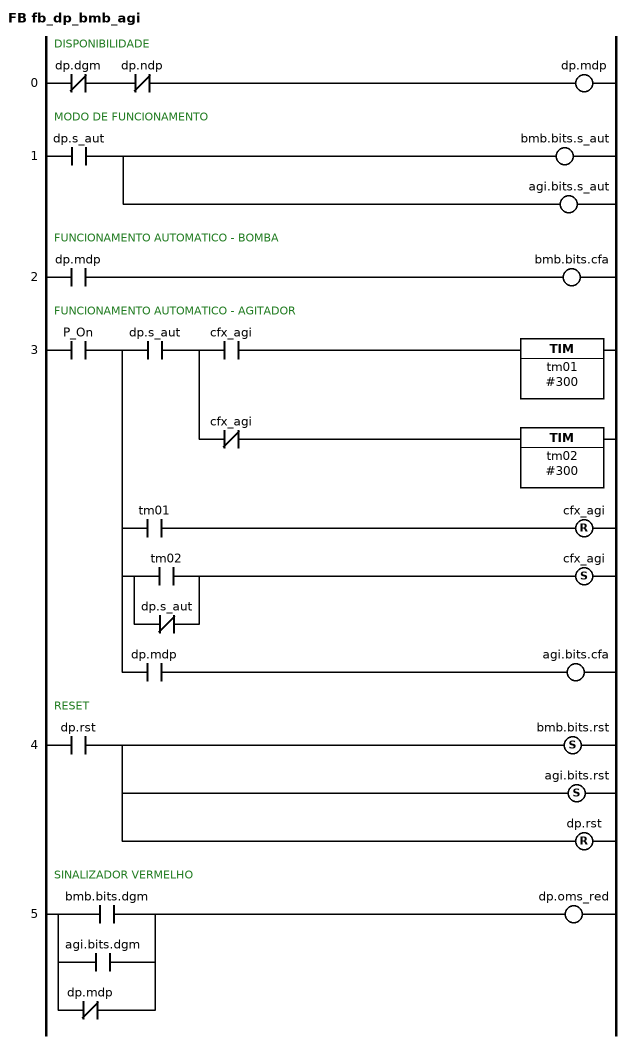
; [picture p24: FB fb_dp_bmb_agi, rungs 0-5]
; rung 0: DISPONIBILIDADE
LDNOT dp.dgm
ANDNOT dp.ndp
OUT dp.mdp
; rung 1: MODO DE FUNCIONAMENTO
LD dp.s_aut
OUT bmb.bits.s_aut
OUT agi.bits.s_aut
; rung 2: FUNCIONAMENTO AUTOMATICO - BOMBA
LD dp.mdp
OUT bmb.bits.cfa
; rung 3: FUNCIONAMENTO AUTOMATICO - AGITADOR
LD P_On
OUT TR0
AND dp.s_aut
OUT TR1
AND cfx_agi
TIM tm01 #300
LD TR1
ANDNOT cfx_agi
TIM tm02 #300
LD TR0
AND tm01
RSET cfx_agi
LD TR0
LD tm02
ORNOT dp.s_aut
ANDLD
SET cfx_agi
LD TR0
AND dp.mdp
OUT agi.bits.cfa
; rung 4: RESET
LD dp.rst
SET bmb.bits.rst
SET agi.bits.rst
RSET dp.rst
; rung 5: SINALIZADOR VERMELHO
LD bmb.bits.dgm
OR agi.bits.dgm
ORNOT dp.mdp
OUT dp.oms_red

## Function block fb_dp_pss_agi_vlv
; FUNÇÃO DEPOSITO DE PRODUTO COM PRESSORIZAÇÃO/AGITADOR/VALVULA - Executa o funcionamento de um deposito de produto constituido por pressorização, um agitador e uma valvula.
VAR_IN_OUT
  dp : s_deposito_p;  (* Dados do deposito *)
  pss : s_equip;  (* Dados da pressorização *)
  agi : s_equip;  (* Dados do agitador *)
  vlv : s_equip;  (* Dados da válvula *)
END_VAR
VAR
  tm01 : TIMER;
  tm02 : TIMER;
  cfx_agi : BOOL;
END_VAR

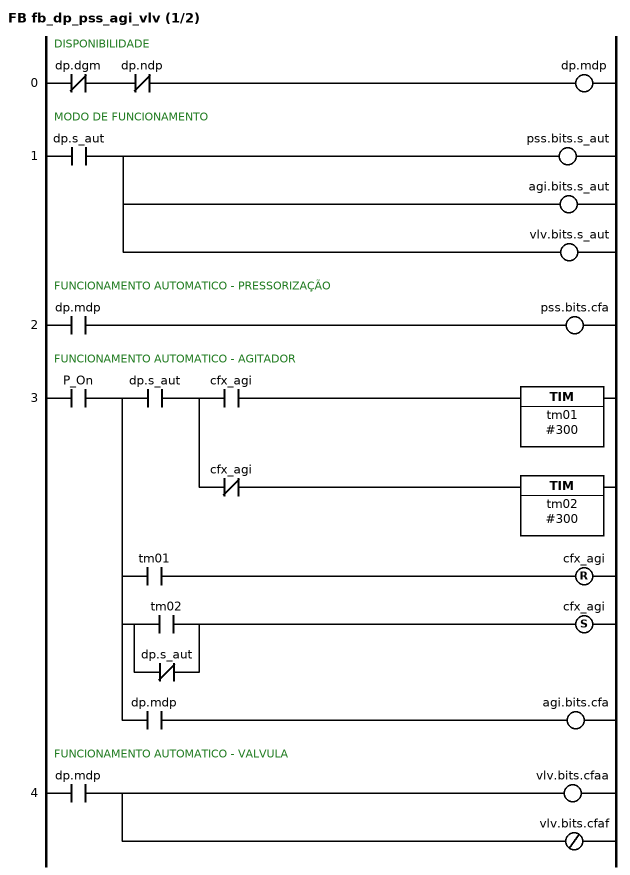
; rung 0: DISPONIBILIDADE
LDNOT dp.dgm
ANDNOT dp.ndp
OUT dp.mdp
; rung 1: MODO DE FUNCIONAMENTO
LD dp.s_aut
OUT pss.bits.s_aut
OUT agi.bits.s_aut
OUT vlv.bits.s_aut
; rung 2: FUNCIONAMENTO AUTOMATICO - PRESSORIZAÇÃO
LD dp.mdp
OUT pss.bits.cfa
; rung 3: FUNCIONAMENTO AUTOMATICO - AGITADOR
LD P_On
OUT TR0
AND dp.s_aut
OUT TR1
AND cfx_agi
TIM tm01 #300
LD TR1
ANDNOT cfx_agi
TIM tm02 #300
LD TR0
AND tm01
RSET cfx_agi
LD TR0
LD tm02
ORNOT dp.s_aut
ANDLD
SET cfx_agi
LD TR0
AND dp.mdp
OUT agi.bits.cfa
; rung 4: FUNCIONAMENTO AUTOMATICO - VALVULA
LD dp.mdp
OUT vlv.bits.cfaa
OUTNOT vlv.bits.cfaf

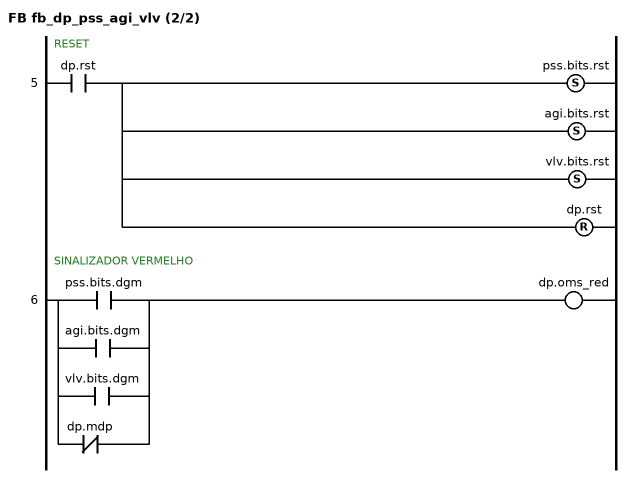
; rung 5: RESET
LD dp.rst
SET pss.bits.rst
SET agi.bits.rst
SET vlv.bits.rst
RSET dp.rst
; rung 6: SINALIZADOR VERMELHO
LD pss.bits.dgm
OR agi.bits.dgm
OR vlv.bits.dgm
ORNOT dp.mdp
OUT dp.oms_red

## Function block fb_eq_bomba
; FUNÇÃO BOMBA - Controlo de uma maquina tipo bomba.
VAR_IN_OUT
  bmb : s_equip;  (* Dados do motor *)
END_VAR
VAR
  tm01 : TIMER;
  tm02 : TIMER;
  ct01 : COUNTER;
  tm_b_x : DINT;
END_VAR

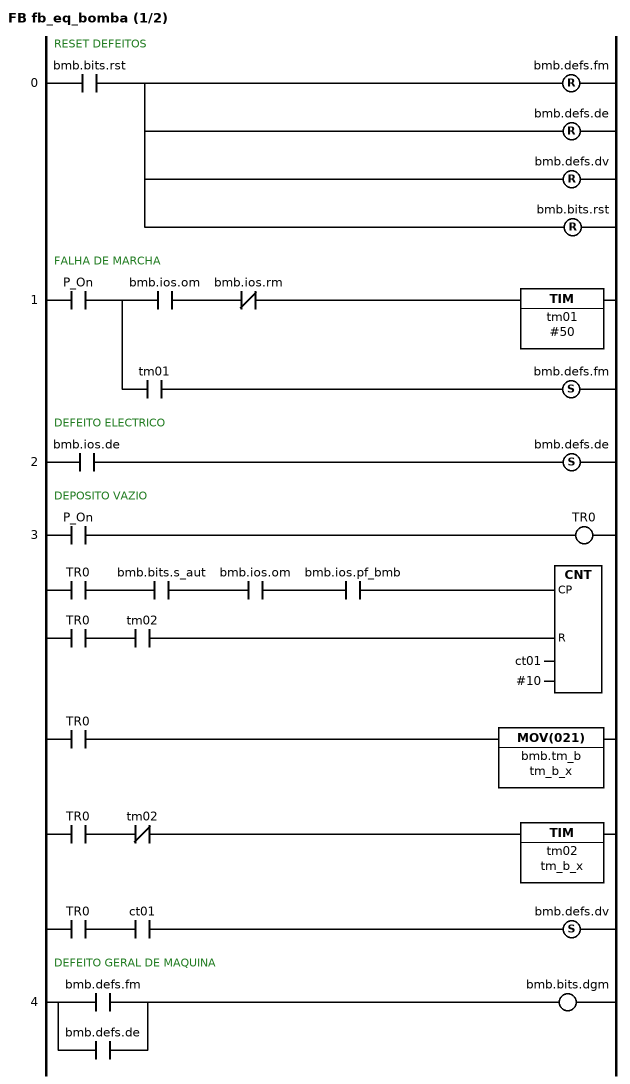
; rung 0: RESET DEFEITOS
LD bmb.bits.rst
RSET bmb.defs.fm
RSET bmb.defs.de
RSET bmb.defs.dv
RSET bmb.bits.rst
; rung 1: FALHA DE MARCHA
LD P_On
OUT TR0
AND bmb.ios.om
ANDNOT bmb.ios.rm
TIM tm01 #50
LD TR0
AND tm01
SET bmb.defs.fm
; rung 2: DEFEITO ELECTRICO
LD bmb.ios.de
SET bmb.defs.de
; rung 3: DEPOSITO VAZIO
LD P_On
OUT TR0
LD TR0
AND bmb.bits.s_aut
AND bmb.ios.om
AND bmb.ios.pf_bmb
LD TR0
AND tm02
CNT ct01 #10
LD TR0
MOV(021) bmb.tm_b tm_b_x
LD TR0
ANDNOT tm02
TIM tm02 tm_b_x
LD TR0
AND ct01
SET bmb.defs.dv
; rung 4: DEFEITO GERAL DE MAQUINA
LD bmb.defs.fm
OR bmb.defs.de
OUT bmb.bits.dgm

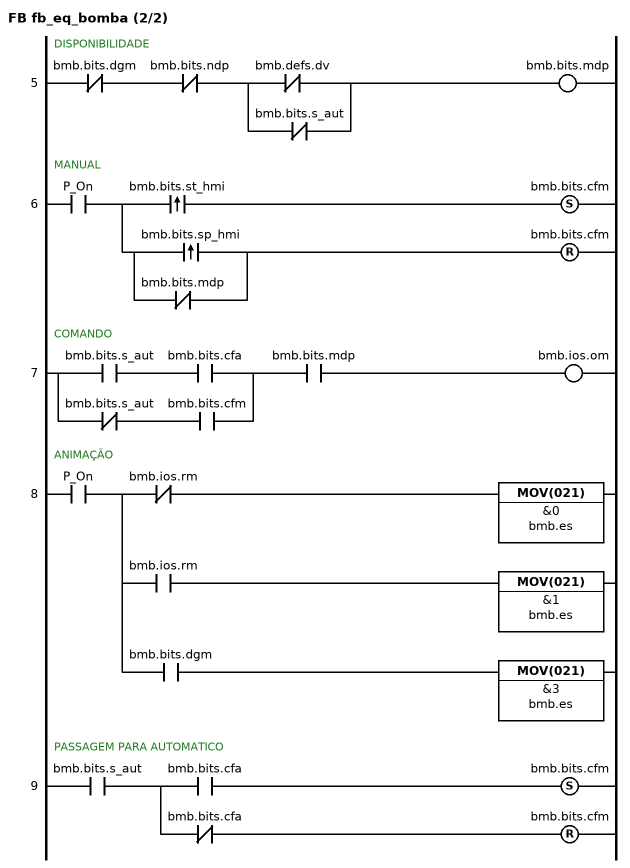
; rung 5: DISPONIBILIDADE
LDNOT bmb.bits.dgm
ANDNOT bmb.bits.ndp
LDNOT bmb.defs.dv
ORNOT bmb.bits.s_aut
ANDLD
OUT bmb.bits.mdp
; rung 6: MANUAL
LD P_On
OUT TR0
@AND bmb.bits.st_hmi
SET bmb.bits.cfm
LD TR0
@LD bmb.bits.sp_hmi
ORNOT bmb.bits.mdp
ANDLD
RSET bmb.bits.cfm
; rung 7: COMANDO
LD bmb.bits.s_aut
AND bmb.bits.cfa
LDNOT bmb.bits.s_aut
AND bmb.bits.cfm
ORLD
AND bmb.bits.mdp
OUT bmb.ios.om
; rung 8: ANIMAÇÃO
LD P_On
OUT TR0
ANDNOT bmb.ios.rm
MOV(021) &0 bmb.es
LD TR0
AND bmb.ios.rm
MOV(021) &1 bmb.es
LD TR0
AND bmb.bits.dgm
MOV(021) &3 bmb.es
; rung 9: PASSAGEM PARA AUTOMATICO
LD bmb.bits.s_aut
OUT TR0
AND bmb.bits.cfa
SET bmb.bits.cfm
LD TR0
ANDNOT bmb.bits.cfa
RSET bmb.bits.cfm

## Function block fb_eq_motor
; FUNÇÃO MOTOR - Controlo de uma maquina tipo motor.
VAR_IN_OUT
  mot : s_equip;  (* Dados do motor *)
END_VAR
VAR
  tm01 : TIMER;
END_VAR

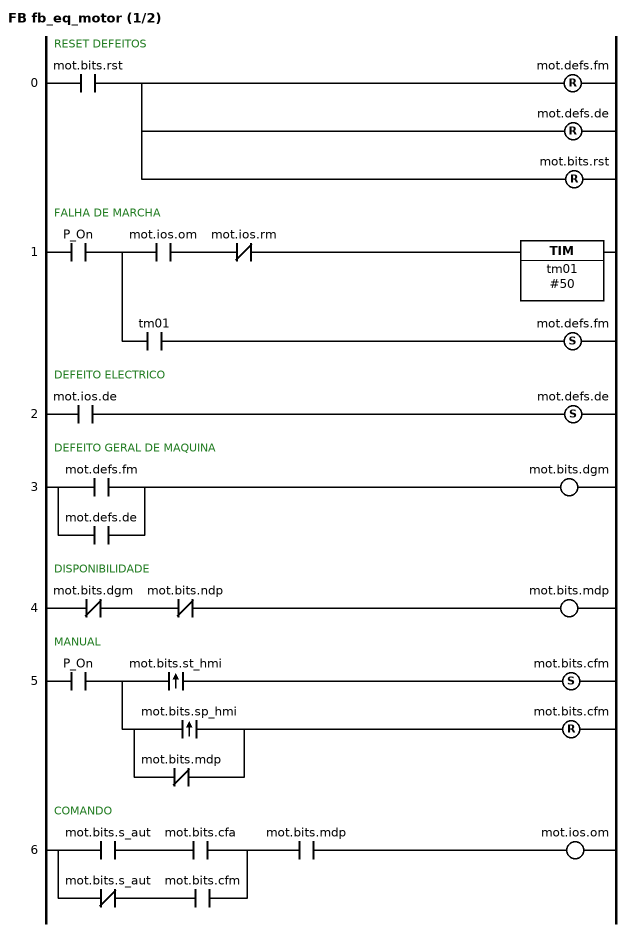
; rung 0: RESET DEFEITOS
LD mot.bits.rst
RSET mot.defs.fm
RSET mot.defs.de
RSET mot.bits.rst
; rung 1: FALHA DE MARCHA
LD P_On
OUT TR0
AND mot.ios.om
ANDNOT mot.ios.rm
TIM tm01 #50
LD TR0
AND tm01
SET mot.defs.fm
; rung 2: DEFEITO ELECTRICO
LD mot.ios.de
SET mot.defs.de
; rung 3: DEFEITO GERAL DE MAQUINA
LD mot.defs.fm
OR mot.defs.de
OUT mot.bits.dgm
; rung 4: DISPONIBILIDADE
LDNOT mot.bits.dgm
ANDNOT mot.bits.ndp
OUT mot.bits.mdp
; rung 5: MANUAL
LD P_On
OUT TR0
@AND mot.bits.st_hmi
SET mot.bits.cfm
LD TR0
@LD mot.bits.sp_hmi
ORNOT mot.bits.mdp
ANDLD
RSET mot.bits.cfm
; rung 6: COMANDO
LD mot.bits.s_aut
AND mot.bits.cfa
LDNOT mot.bits.s_aut
AND mot.bits.cfm
ORLD
AND mot.bits.mdp
OUT mot.ios.om

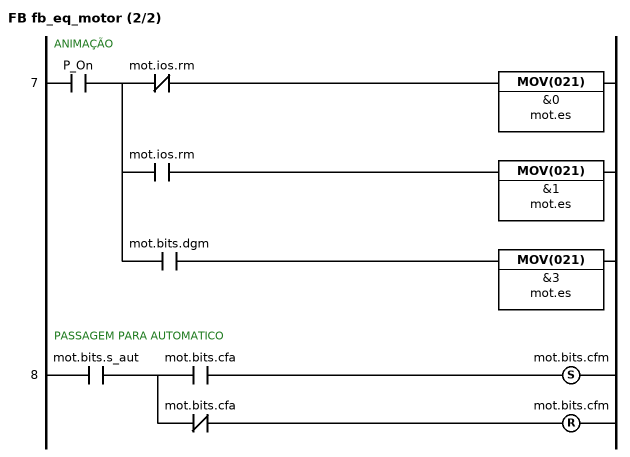
; rung 7: ANIMAÇÃO
LD P_On
OUT TR0
ANDNOT mot.ios.rm
MOV(021) &0 mot.es
LD TR0
AND mot.ios.rm
MOV(021) &1 mot.es
LD TR0
AND mot.bits.dgm
MOV(021) &3 mot.es
; rung 8: PASSAGEM PARA AUTOMATICO
LD mot.bits.s_aut
OUT TR0
AND mot.bits.cfa
SET mot.bits.cfm
LD TR0
ANDNOT mot.bits.cfa
RSET mot.bits.cfm

## Function block fb_eq_press
; FUNÇÃO PRESSORIZAR - Controlo de uma maquina tipo motor.
VAR_IN_OUT
  press : s_equip;  (* Dados da presseorização *)
END_VAR
VAR
  tm01 : TIMER;
END_VAR

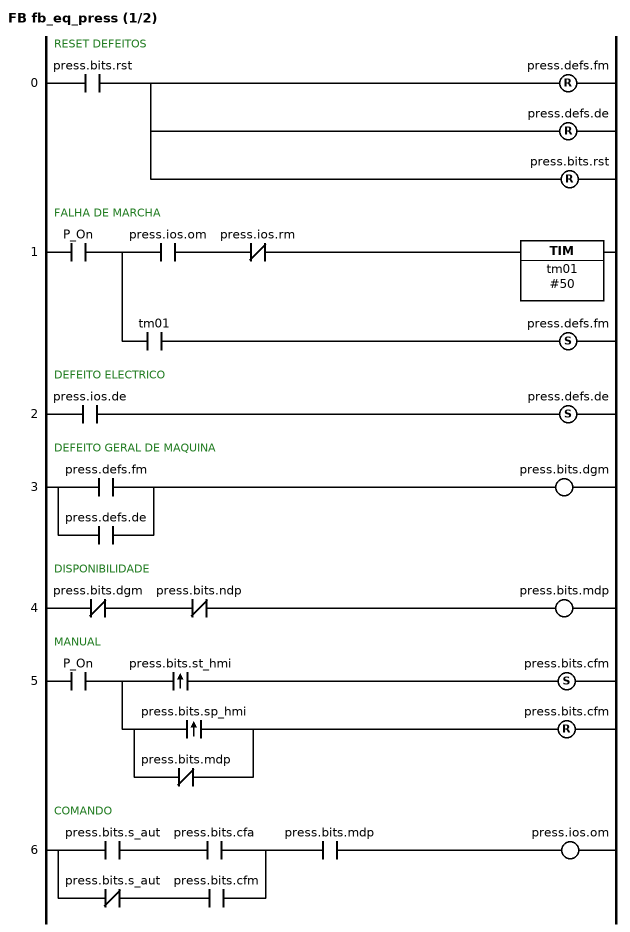
; rung 0: RESET DEFEITOS
LD press.bits.rst
RSET press.defs.fm
RSET press.defs.de
RSET press.bits.rst
; rung 1: FALHA DE MARCHA
LD P_On
OUT TR0
AND press.ios.om
ANDNOT press.ios.rm
TIM tm01 #50
LD TR0
AND tm01
SET press.defs.fm
; rung 2: DEFEITO ELECTRICO
LD press.ios.de
SET press.defs.de
; rung 3: DEFEITO GERAL DE MAQUINA
LD press.defs.fm
OR press.defs.de
OUT press.bits.dgm
; rung 4: DISPONIBILIDADE
LDNOT press.bits.dgm
ANDNOT press.bits.ndp
OUT press.bits.mdp
; rung 5: MANUAL
LD P_On
OUT TR0
@AND press.bits.st_hmi
SET press.bits.cfm
LD TR0
@LD press.bits.sp_hmi
ORNOT press.bits.mdp
ANDLD
RSET press.bits.cfm
; rung 6: COMANDO
LD press.bits.s_aut
AND press.bits.cfa
LDNOT press.bits.s_aut
AND press.bits.cfm
ORLD
AND press.bits.mdp
OUT press.ios.om

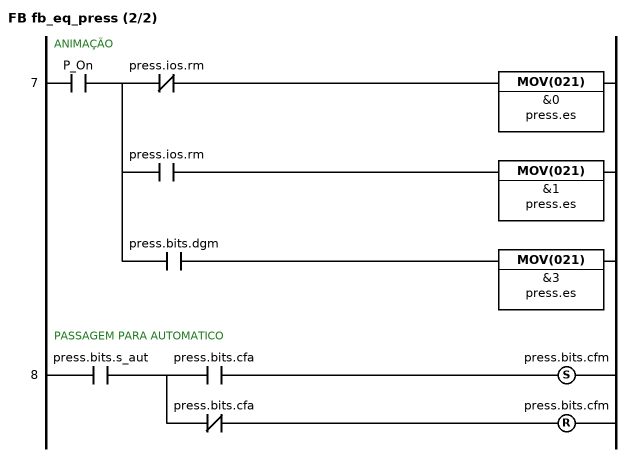
; rung 7: ANIMAÇÃO
LD P_On
OUT TR0
ANDNOT press.ios.rm
MOV(021) &0 press.es
LD TR0
AND press.ios.rm
MOV(021) &1 press.es
LD TR0
AND press.bits.dgm
MOV(021) &3 press.es
; rung 8: PASSAGEM PARA AUTOMATICO
LD press.bits.s_aut
OUT TR0
AND press.bits.cfa
SET press.bits.cfm
LD TR0
ANDNOT press.bits.cfa
RSET press.bits.cfm

## Function block fb_eq_valvula
; FUNÇÃO VALVULA - Controlo de uma maquina tipo valvula.
VAR_IN_OUT
  valv : s_equip;  (* Dados da valvula *)
END_VAR
VAR
  tm01 : TIMER;
  tm02 : TIMER;
END_VAR

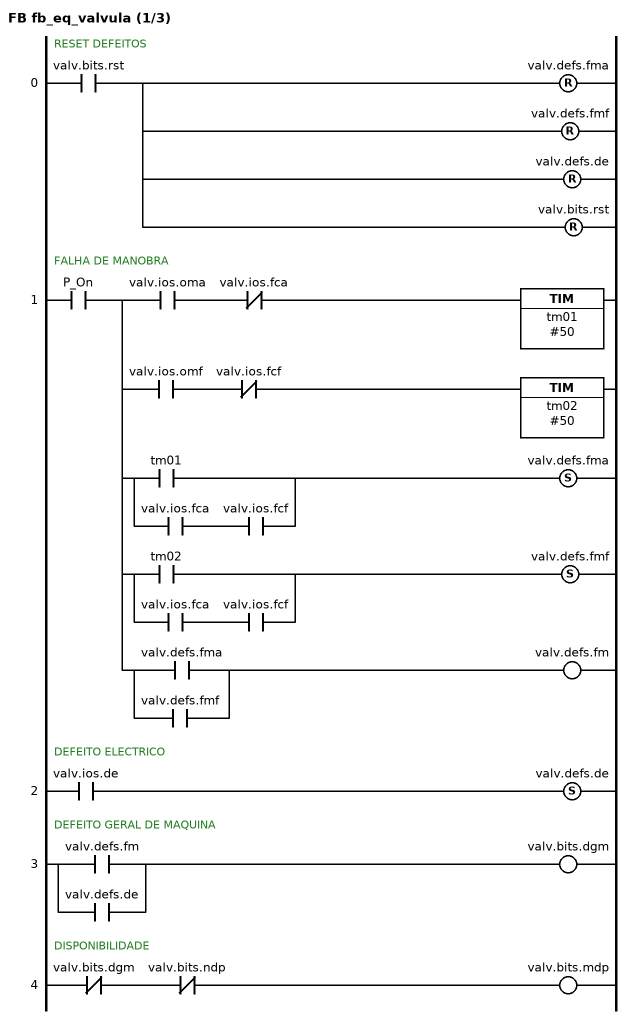
; rung 0: RESET DEFEITOS
LD valv.bits.rst
RSET valv.defs.fma
RSET valv.defs.fmf
RSET valv.defs.de
RSET valv.bits.rst
; rung 1: FALHA DE MANOBRA
LD P_On
OUT TR0
AND valv.ios.oma
ANDNOT valv.ios.fca
TIM tm01 #50
LD TR0
AND valv.ios.omf
ANDNOT valv.ios.fcf
TIM tm02 #50
LD TR0
LD tm01
LD valv.ios.fca
AND valv.ios.fcf
ORLD
ANDLD
SET valv.defs.fma
LD TR0
LD tm02
LD valv.ios.fca
AND valv.ios.fcf
ORLD
ANDLD
SET valv.defs.fmf
LD TR0
LD valv.defs.fma
OR valv.defs.fmf
ANDLD
OUT valv.defs.fm
; rung 2: DEFEITO ELECTRICO
LD valv.ios.de
SET valv.defs.de
; rung 3: DEFEITO GERAL DE MAQUINA
LD valv.defs.fm
OR valv.defs.de
OUT valv.bits.dgm
; rung 4: DISPONIBILIDADE
LDNOT valv.bits.dgm
ANDNOT valv.bits.ndp
OUT valv.bits.mdp

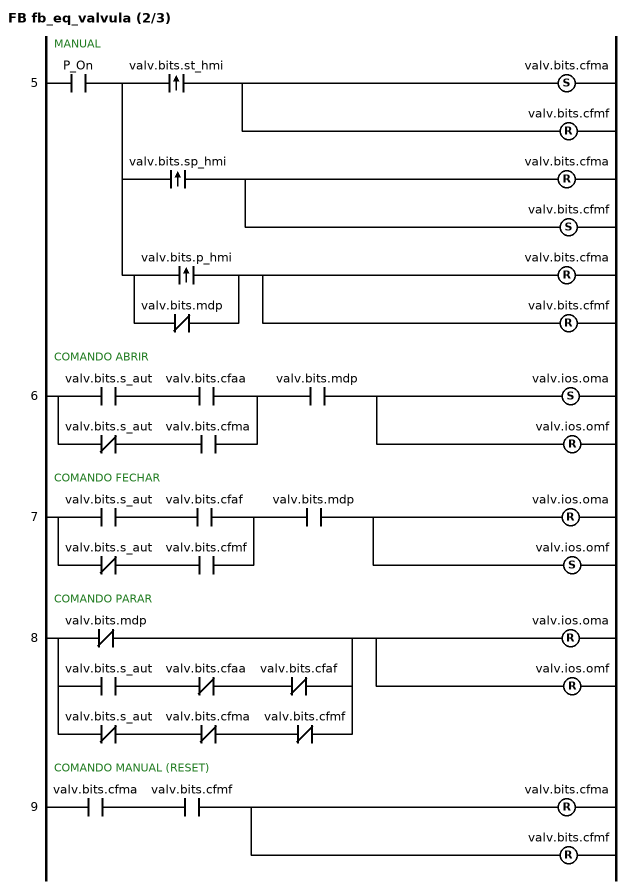
; rung 5: MANUAL
LD P_On
OUT TR0
@AND valv.bits.st_hmi
SET valv.bits.cfma
RSET valv.bits.cfmf
LD TR0
@AND valv.bits.sp_hmi
RSET valv.bits.cfma
SET valv.bits.cfmf
LD TR0
@LD valv.bits.p_hmi
ORNOT valv.bits.mdp
ANDLD
RSET valv.bits.cfma
RSET valv.bits.cfmf
; rung 6: COMANDO ABRIR
LD valv.bits.s_aut
AND valv.bits.cfaa
LDNOT valv.bits.s_aut
AND valv.bits.cfma
ORLD
AND valv.bits.mdp
SET valv.ios.oma
RSET valv.ios.omf
; rung 7: COMANDO FECHAR
LD valv.bits.s_aut
AND valv.bits.cfaf
LDNOT valv.bits.s_aut
AND valv.bits.cfmf
ORLD
AND valv.bits.mdp
RSET valv.ios.oma
SET valv.ios.omf
; rung 8: COMANDO PARAR
LDNOT valv.bits.mdp
LD valv.bits.s_aut
ANDNOT valv.bits.cfaa
ANDNOT valv.bits.cfaf
ORLD
LDNOT valv.bits.s_aut
ANDNOT valv.bits.cfma
ANDNOT valv.bits.cfmf
ORLD
RSET valv.ios.oma
RSET valv.ios.omf
; rung 9: COMANDO MANUAL (RESET)
LD valv.bits.cfma
AND valv.bits.cfmf
RSET valv.bits.cfma
RSET valv.bits.cfmf

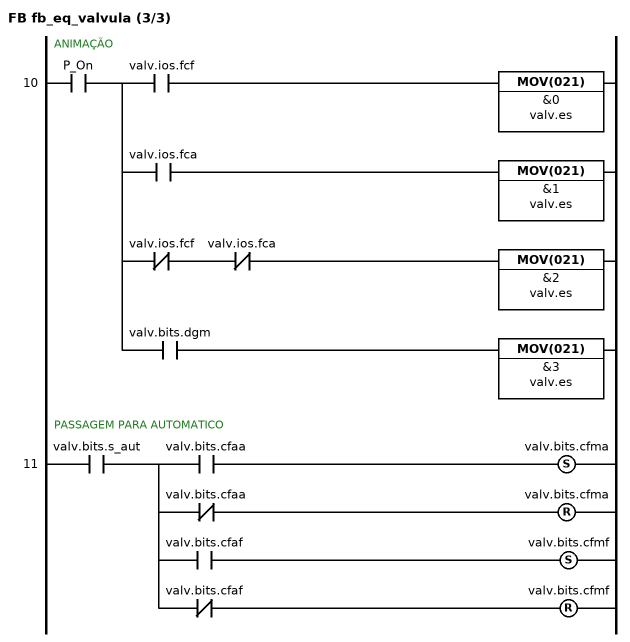
; rung 10: ANIMAÇÃO
LD P_On
OUT TR0
AND valv.ios.fcf
MOV(021) &0 valv.es
LD TR0
AND valv.ios.fca
MOV(021) &1 valv.es
LD TR0
ANDNOT valv.ios.fcf
ANDNOT valv.ios.fca
MOV(021) &2 valv.es
LD TR0
AND valv.bits.dgm
MOV(021) &3 valv.es
; rung 11: PASSAGEM PARA AUTOMATICO
LD valv.bits.s_aut
OUT TR0
AND valv.bits.cfaa
SET valv.bits.cfma
LD TR0
ANDNOT valv.bits.cfaa
RSET valv.bits.cfma
LD TR0
AND valv.bits.cfaf
SET valv.bits.cfmf
LD TR0
ANDNOT valv.bits.cfaf
RSET valv.bits.cfmf

## Function block fb_inj_caudal
; FUNÇÃO CAUDALIMETRO - Caudalimetro local/remoto
VAR_IN_OUT
  tt : s_caudal;  (* Dados do caudalímetro *)
END_VAR
VAR
  tt_rem_d : REAL;  (* Diferença de totalização *)
  tm01 : TIMER;
  tm02 : TIMER;
  ct01 : COUNTER;
END_VAR

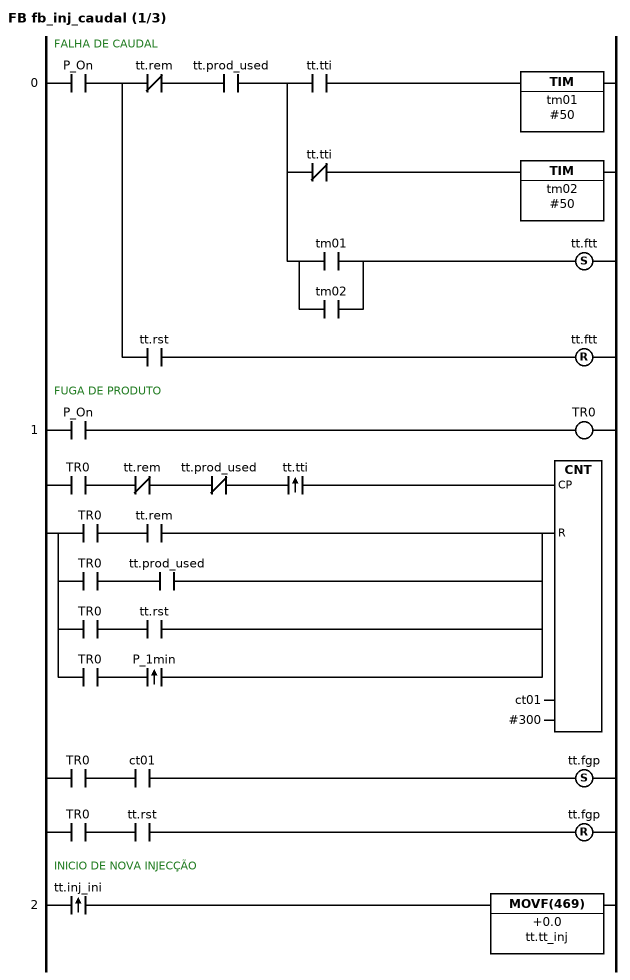
; rung 0: FALHA DE CAUDAL
LD P_On
OUT TR0
ANDNOT tt.rem
AND tt.prod_used
OUT TR1
AND tt.tti
TIM tm01 #50
LD TR1
ANDNOT tt.tti
TIM tm02 #50
LD TR1
LD tm01
OR tm02
ANDLD
SET tt.ftt
LD TR0
AND tt.rst
RSET tt.ftt
; rung 1: FUGA DE PRODUTO
LD P_On
OUT TR0
LD TR0
ANDNOT tt.rem
ANDNOT tt.prod_used
@AND tt.tti
LD TR0
AND tt.rem
LD TR0
AND tt.prod_used
ORLD
LD TR0
AND tt.rst
ORLD
LD TR0
@AND P_1min
ORLD
CNT ct01 #300
LD TR0
AND ct01
SET tt.fgp
LD TR0
AND tt.rst
RSET tt.fgp
; rung 2: INICIO DE NOVA INJECÇÃO
@LD tt.inj_ini
MOVF(469) +0.0 tt.tt_inj

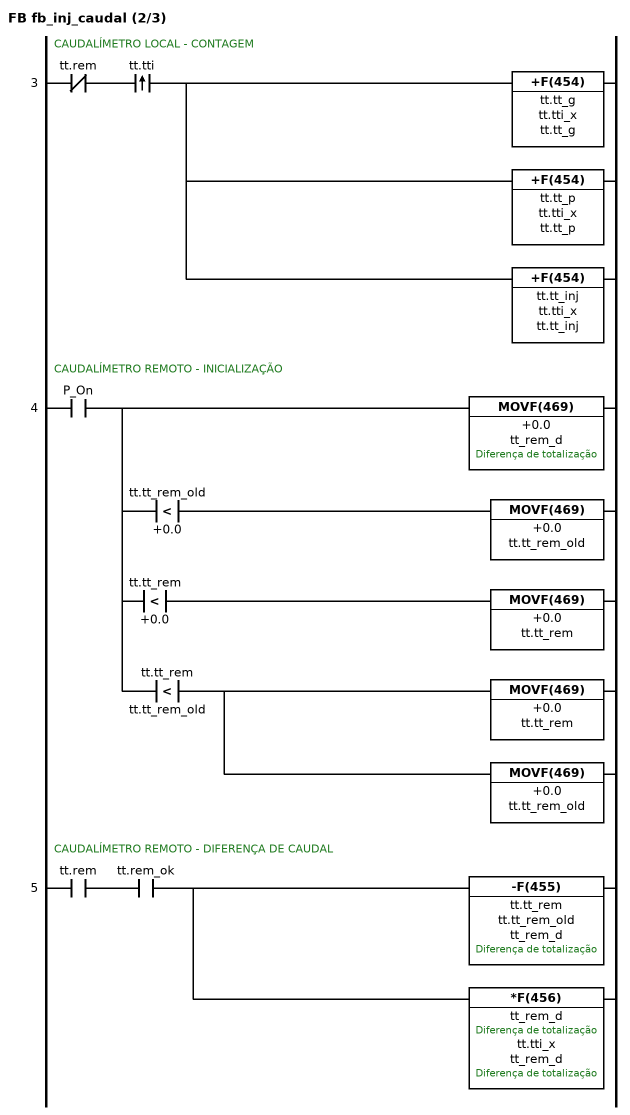
; rung 3: CAUDALÍMETRO LOCAL - CONTAGEM
LDNOT tt.rem
@AND tt.tti
+F(454) tt.tt_g tt.tti_x tt.tt_g
+F(454) tt.tt_p tt.tti_x tt.tt_p
+F(454) tt.tt_inj tt.tti_x tt.tt_inj
; rung 4: CAUDALÍMETRO REMOTO - INICIALIZAÇÃO
LD P_On
OUT TR0
MOVF(469) +0.0 tt_rem_d  ; Diferença de totalização
AND<F(331) tt.tt_rem_old +0.0
MOVF(469) +0.0 tt.tt_rem_old
LD TR0
AND<F(331) tt.tt_rem +0.0
MOVF(469) +0.0 tt.tt_rem
LD TR0
AND<F(331) tt.tt_rem tt.tt_rem_old
MOVF(469) +0.0 tt.tt_rem
MOVF(469) +0.0 tt.tt_rem_old
; rung 5: CAUDALÍMETRO REMOTO - DIFERENÇA DE CAUDAL
LD tt.rem
AND tt.rem_ok
-F(455) tt.tt_rem tt.tt_rem_old tt_rem_d  ; Diferença de totalização
*F(456) tt_rem_d tt.tti_x tt_rem_d  ; Diferença de totalização

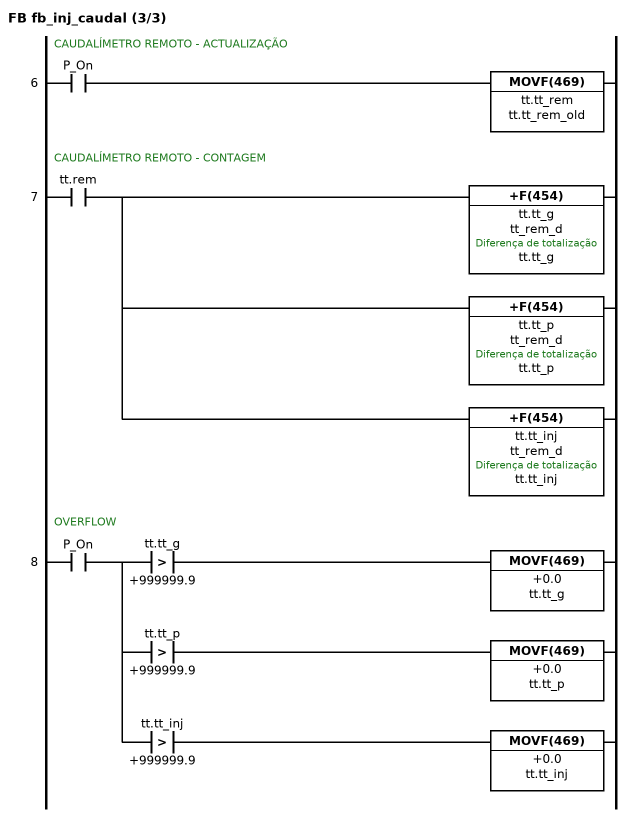
; rung 6: CAUDALÍMETRO REMOTO - ACTUALIZAÇÃO
LD P_On
MOVF(469) tt.tt_rem tt.tt_rem_old
; rung 7: CAUDALÍMETRO REMOTO - CONTAGEM
LD tt.rem
+F(454) tt.tt_g tt_rem_d tt.tt_g  ; Diferença de totalização
+F(454) tt.tt_p tt_rem_d tt.tt_p  ; Diferença de totalização
+F(454) tt.tt_inj tt_rem_d tt.tt_inj  ; Diferença de totalização
; rung 8: OVERFLOW
LD P_On
OUT TR0
AND>F(333) tt.tt_g +999999.9
MOVF(469) +0.0 tt.tt_g
LD TR0
AND>F(333) tt.tt_p +999999.9
MOVF(469) +0.0 tt.tt_p
LD TR0
AND>F(333) tt.tt_inj +999999.9
MOVF(469) +0.0 tt.tt_inj

## Function block fb_prod_ok
; FUNÇÃO PRODUTO OK - Verifica se o produto não está a ser doseado para outra maquina, e autoriza a maquina a dosear (caudalimetros comuns).
VAR_IN_OUT
  m_prod_in : ARRAY[0..9] OF INT;  (* Produto pedido *)
  m_prod_out : ARRAY[0..9] OF INT;  (* Produto autorizado *)
  prod_used : ARRAY[0..9] OF BOOL;  (* Produto em uso *)
END_VAR
VAR
  i : INT;
  k : INT;
  ok : BOOL;
END_VAR
(*Verificar que maquinas deixaram de pedir produto*)
FOR i:= 0 TO 9 DO
	IF m_prod_in[i]=0 THEN
		m_prod_out[i]:= 0;
	END_IF;
END_FOR;

(*Atribuir produto às maquinas*)
FOR i:= 0 TO 9 DO
	ok:= TRUE;
	FOR k:= 0 TO 9 DO
		IF k<>i AND m_prod_out[k]=m_prod_in[i] THEN
			ok:= FALSE;
		END_IF;
	END_FOR;
	IF ok=TRUE THEN
		m_prod_out[i]:= m_prod_in[i];
	ELSE
		m_prod_out[i]:= 0;
	END_IF;
END_FOR;

(*Verifica se o produto está em uso*)
FOR i:= 0 TO 9 DO
	prod_used[i]:= FALSE;
	FOR k:= 0 TO 9 DO
		IF m_prod_out[k]-1= i THEN
			prod_used[i]:= TRUE;
		END_IF;
	END_FOR;
END_FOR;

## Function block fb_relogio
VAR_IN_OUT
  relogio : s_relogio;  (* Dados do relogio *)
END_VAR
VAR
  data_hora : LWORD;
END_VAR

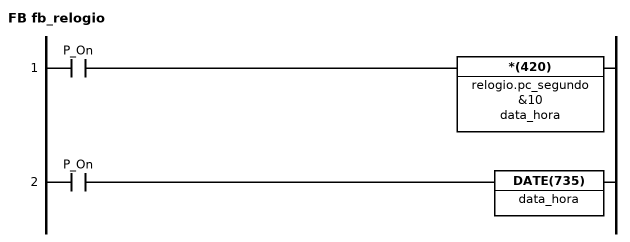
; rung 1
LD P_On
*(420) relogio.pc_segundo &10 data_hora
; rung 2
LD P_On
DATE(735) data_hora